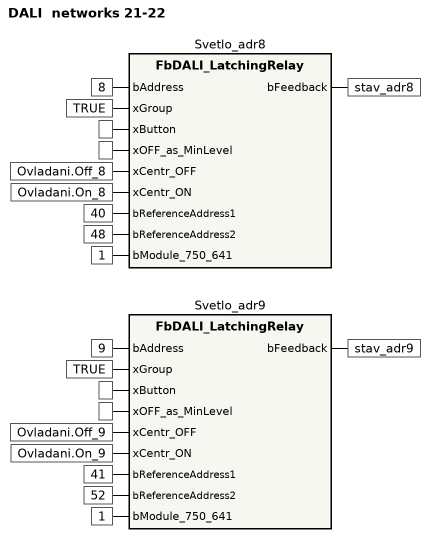
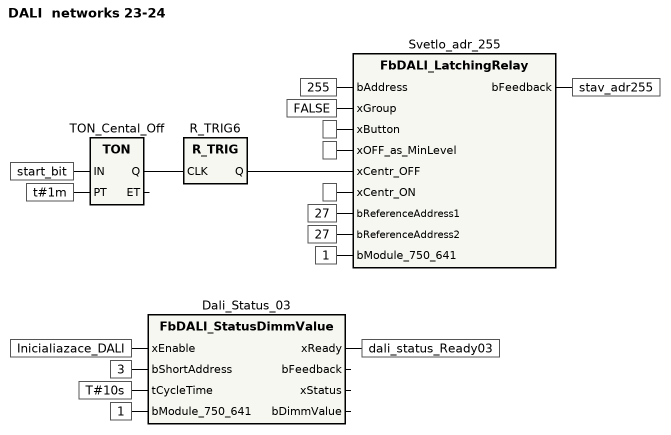
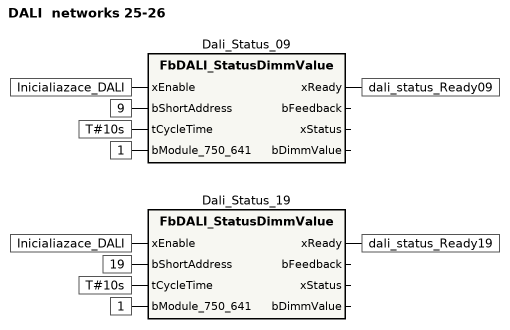
_FBD_ (* Function Block Diagram *)
NETWORK 1
	D_M:FbDALI_Joblist(bModule_750_641: 1)
NETWORK 2
	???:DALI_Config()
NETWORK 3
	Trojklik_Fagule_OUT13:Trojklik(TL1: , TL2: , TL3: , TL4: OR(TL10, TL10s, TL10p), TL5: , TL6: , RESET_Rezim_1klik: OR(OP_reset5, OP_reset1), RESET_Rezim_2klik: , RESET_Rezim_3klik: , RESET_Rezim_OUT15: , RESET_Rezim_OUT16: , Pocet_kliku_MAX: 1, AUT_vyp: FALSE, cas_vypnuti: t#30m, Rezim_1klik_OFF_ON => KA01, Rezim_OUT15_OFF_ON => KA13)
NETWORK 4
	ka13pink:TP(IN: ka13cas:TON(IN: KA13, PT: casvensvetel), PT: t#1s) => TL10p
NETWORK 5
	Fb_LatchingRelay1:Fb_LatchingRelay(Fb_ShortLong1:Fb_ShortLong(OR(TL06, TL06s, TL06p), 10, 1, 1, out 2 => KratkyKlikA), , , ) => KA15
NETWORK 6
	ka15pink:TP(IN: ka15cas:TON(IN: KA15, PT: casvensvetel), PT: t#1s) => TL06p
NETWORK 7
	Fb_LatchingRelay2:Fb_LatchingRelay(Fb_ShortLong2:Fb_ShortLong(OR(TL05, TL05s, TL04, TL05p), 10, 1, 1, out 2 => KratkyKlikB), , , ) => KA16
NETWORK 8
	ka16pink:TP(IN: ka16cas:TON(IN: KA16, PT: casvensvetel), PT: t#1s) => TL05p
NETWORK 9
	Fb_ShortLong3:Fb_ShortLong(OR(TL03, TL01, TL01s, TL02), 10, 1, 1, out 2 => KratkyKlikC)
NETWORK 10
	OR(KratkyKlikA, KratkyKlikB, KratkyKlikC) => KratkyKlik
NETWORK 11
	CTU1:CTU(CU: AND(TP1:TP(IN: KratkyKlik, PT: CasNaKlik), R_TRIG1:R_TRIG(CLK: KratkyKlik)), RESET: R_TRIG2:R_TRIG(CLK: Zhasni1.xPresunuto), PV: 3, CV => STAV)
NETWORK 12
	Zhasni1:Zhasni(wIn: STAV, xPresun: F_TRIG3:F_TRIG(CLK: TP1.Q))
NETWORK 13
	Svetlo_adr1:FbDALI_LatchingRelay(bAddress: 1, xGroup: TRUE, xButton: , xOFF_as_MinLevel: , xCentr_OFF: Zhasni1.xoffOUT1, xCentr_ON: Zhasni1.xonOUT1, bReferenceAddress1: 3, bReferenceAddress2: 9, bModule_750_641: 1) => stav_adr1
NETWORK 14
	Svetlo_adr2:FbDALI_LatchingRelay(bAddress: 2, xGroup: TRUE, xButton: , xOFF_as_MinLevel: , xCentr_OFF: Zhasni1.xoffOUT2, xCentr_ON: Zhasni1.xonOUT2, bReferenceAddress1: 17, bReferenceAddress2: 17, bModule_750_641: 1) => stav_adr2
NETWORK 15
	Svetlo_adr3:FbDALI_LatchingRelay(bAddress: 3, xGroup: TRUE, xButton: , xOFF_as_MinLevel: , xCentr_OFF: Zhasni1.xoffOUT3, xCentr_ON: Zhasni1.xonOUT3, bReferenceAddress1: 27, bReferenceAddress2: 27, bModule_750_641: 1) => stav_adr3
NETWORK 16
	Svetlo_adr4:FbDALI_DimmSingleButton(bAddress: 4, xGroup: TRUE, xButton: OR(TL09, TL09s), bSwitchOnLevel: hodnota_po_zapnuti_prodejna, xOFF_at_MinLevel: povolit_vypnuti_pri_minimum, xOFF_as_MinLevel: , bFadeRate: rychlost_zneny, tShortPushButton: co_je_kratky_a_dlouhy_stisk, bReferenceaddress1: 29, bReferenceaddress2: 30, bModule_750_641: 1) => stav_adr4
NETWORK 17
	Svetlo_adr5:FbDALI_LatchingRelay(bAddress: 5, xGroup: TRUE, xButton: OR(TL12, FALSE), xOFF_as_MinLevel: , xCentr_OFF: , xCentr_ON: , bReferenceAddress1: 37, bReferenceAddress2: 45, bModule_750_641: 1) => stav_adr5
NETWORK 18
	Svetlo_adr6:FbDALI_LatchingRelay(bAddress: 6, xGroup: TRUE, xButton: OR(TL13, FALSE), xOFF_as_MinLevel: , xCentr_OFF: , xCentr_ON: , bReferenceAddress1: 47, bReferenceAddress2: 49, bModule_750_641: 1) => stav_adr6
NETWORK 19
	Ovladani:Ovladani_7_8_9(xVstup: OR(TL11, FALSE), rCidlo: Cidlo, rUroven1: Uroven1, rUroven2: Uroven2, tZpozdeniCidla: DWORD_TO_TIME(MUL(ZpozdeniCidla, 60000)))
NETWORK 20
	Svetlo_adr7:FbDALI_LatchingRelay(bAddress: 7, xGroup: TRUE, xButton: , xOFF_as_MinLevel: , xCentr_OFF: Ovladani.Off_7, xCentr_ON: Ovladani.On_7, bReferenceAddress1: 36, bReferenceAddress2: 50, bModule_750_641: 1) => stav_adr7
NETWORK 21
	Svetlo_adr8:FbDALI_LatchingRelay(bAddress: 8, xGroup: TRUE, xButton: , xOFF_as_MinLevel: , xCentr_OFF: Ovladani.Off_8, xCentr_ON: Ovladani.On_8, bReferenceAddress1: 40, bReferenceAddress2: 48, bModule_750_641: 1) => stav_adr8
NETWORK 22
	Svetlo_adr9:FbDALI_LatchingRelay(bAddress: 9, xGroup: TRUE, xButton: , xOFF_as_MinLevel: , xCentr_OFF: Ovladani.Off_9, xCentr_ON: Ovladani.On_9, bReferenceAddress1: 41, bReferenceAddress2: 52, bModule_750_641: 1) => stav_adr9
NETWORK 23 (* Po 1min po restartu dojde k vypnuti vsech svitidel *)
	Svetlo_adr_255:FbDALI_LatchingRelay(bAddress: 255, xGroup: FALSE, xButton: , xOFF_as_MinLevel: , xCentr_OFF: R_TRIG6:R_TRIG(CLK: TON_Cental_Off:TON(IN: start_bit, PT: t#1m)), xCentr_ON: , bReferenceAddress1: 27, bReferenceAddress2: 27, bModule_750_641: 1) => stav_adr255
NETWORK 24
	Dali_Status_03:FbDALI_StatusDimmValue(xEnable: Inicialiazace_DALI, bShortAddress: 3, tCycleTime: T#10s, bModule_750_641: 1) => dali_status_Ready03
NETWORK 25
	Dali_Status_09:FbDALI_StatusDimmValue(xEnable: Inicialiazace_DALI, bShortAddress: 9, tCycleTime: T#10s, bModule_750_641: 1) => dali_status_Ready09
NETWORK 26
	Dali_Status_19:FbDALI_StatusDimmValue(xEnable: Inicialiazace_DALI, bShortAddress: 19, tCycleTime: T#10s, bModule_750_641: 1) => dali_status_Ready19
_END_FBD_
(* the same logic as Structured Text *)
(* Network 1 *)
D_M(bModule_750_641 := 1);
(* Network 2: see the listing above *)
(* Network 3: see the listing above *)
(* Network 4 *)
ka13cas(IN := KA13, PT := casvensvetel);
ka13pink(IN := ka13cas.Q, PT := t#1s);
TL10p := ka13pink.Q;
(* Network 5: see the listing above *)
(* Network 6 *)
ka15cas(IN := KA15, PT := casvensvetel);
ka15pink(IN := ka15cas.Q, PT := t#1s);
TL06p := ka15pink.Q;
(* Network 7: see the listing above *)
(* Network 8 *)
ka16cas(IN := KA16, PT := casvensvetel);
ka16pink(IN := ka16cas.Q, PT := t#1s);
TL05p := ka16pink.Q;
(* Network 9: see the listing above *)
(* Network 10 *)
KratkyKlik := KratkyKlikA OR KratkyKlikB OR KratkyKlikC;
(* Network 11 *)
TP1(IN := KratkyKlik, PT := CasNaKlik);
R_TRIG1(CLK := KratkyKlik);
R_TRIG2(CLK := Zhasni1.xPresunuto);
CTU1(CU := TP1.Q AND R_TRIG1.Q, RESET := R_TRIG2.Q, PV := 3);
STAV := CTU1.CV;
(* Network 12 *)
F_TRIG3(CLK := TP1.Q);
Zhasni1(wIn := STAV, xPresun := F_TRIG3.Q);
(* Network 13: see the listing above *)
(* Network 14: see the listing above *)
(* Network 15: see the listing above *)
(* Network 16: see the listing above *)
(* Network 17: see the listing above *)
(* Network 18: see the listing above *)
(* Network 19: see the listing above *)
(* Network 20: see the listing above *)
(* Network 21: see the listing above *)
(* Network 22: see the listing above *)
(* Network 23: see the listing above *)
(* Network 24 *)
Dali_Status_03(xEnable := Inicialiazace_DALI, bShortAddress := 3, tCycleTime := T#10s, bModule_750_641 := 1);
dali_status_Ready03 := Dali_Status_03.xReady;
(* Network 25 *)
Dali_Status_09(xEnable := Inicialiazace_DALI, bShortAddress := 9, tCycleTime := T#10s, bModule_750_641 := 1);
dali_status_Ready09 := Dali_Status_09.xReady;
(* Network 26 *)
Dali_Status_19(xEnable := Inicialiazace_DALI, bShortAddress := 19, tCycleTime := T#10s, bModule_750_641 := 1);
dali_status_Ready19 := Dali_Status_19.xReady;
END_PROGRAM

(* POU dali/Trojklik, FBD *)
FUNCTION_BLOCK Trojklik
VAR
	TLx_sklad: BOOL;
	Data_platna: BOOL;
	Data_platna_reset: BOOL;
	T_Data_platna: TON;
	T_Data_platna_reset: TON;
	Stisk_kratky: BOOL := FALSE;
	Stisk_dlouhy: BOOL := FALSE;
	Q_stisk_TLx: BOOL;
	T_stisk_TLx: TON;
	F_trig_hr1: F_TRIG;
	R_trig_hr2: R_TRIG;
	TLx_sklad_hr1: BOOL;
	TLx_INT: INT;
	TLx_Citac: CTU;
	SET_stisk_TLx: BOOL;
	SR_stisk_TLx: SR;

	ZAP_VYP_sklad: BOOL;
	mod_1klik: BOOL;
	mod_2klik: BOOL;
	blok: BOOL;
	blok_ZAP_VYP: BOOL;
	T_blok: TON;
	T_blok_ZAP_VYP: TON;
	TP_mode_1klik: TP;

	TP_mode_2klik: TP;

	TP_byl_kratky: TP;
	Q_byl_kratky: BOOL;
	blok_kratky: BOOL;
	mod_3klik: BOOL;
	TP_mode_3klik: TP;

	TP_reset1: TP;
	TP_reset2: TP;
	TP_reset3: TP;
	TLx_zvenku: BOOL;
	T_stisk_TLx_zvenku: TON;
	TLx_sklad_hr1_zvenku: BOOL;
	F_trig_hr1_zvenku: F_TRIG;
	Stisk_kratky_zvenku: BOOL;
	SET_stisk_TLx_zvenku: BOOL;
	Q_byl_kratky_zvenku: BOOL;
	TP_byl_kratky_zvenku: TP;
	Stisk_dlouhy_zvenku: BOOL;
	blok_kratky_zvenku: BOOL;
	TLx_INT_zvenku: INT;
	TLx_Citac_zvenku: CTU;
	Q_stisk_TLx_zvenku: BOOL;
	R_trig_hr2_zvenku: R_TRIG;
	SR_stisk_TLx_zvenku: SR;
	blok_OUT15: BOOL;
	TOF_OUT15_zp: TOF;
	R_trig_OUT15: R_TRIG;
	R_trig_OUT15b: R_TRIG;
	TON_blok_OUT15: TON;
	TON_AUT_stop_OUT15: TON;
	R_trig_OUT16: R_TRIG;
	TOF_OUT16_zp: TOF;
	blok_OUT16: BOOL;
	R_trig_OUT16b: R_TRIG;
	TON_AUT_stop_OUT16: TON;
	TON_blok_OUT16: TON;
	T_max: TON;
	Q_T_MAX: BOOL;
	TP_T_max: TP;
	Aktivni_TL1: BOOL;
	Aktivni_TL2: BOOL;
	Aktivni_TL3: BOOL;
	Aktivni_TL4: BOOL;
	Aktivni_TL5: BOOL;
	Aktivni_TL6: BOOL;
	T_vypnuti_ukonceno: TP;
	Q_vypnuti_ukonceno: BOOL;
	F_trig_1klik: F_TRIG;
	F_trig_2klik: F_TRIG;
	F_trig_3klik: F_TRIG;
	tp_1klik_vyp: TP;
	f_trig_1klik_vyp: F_TRIG;
	tp_2klik_vyp: TP;
	f_trig_2klik_vyp: F_TRIG;
	f_trig_3klik_vyp: F_TRIG;
	tp_3klik_vyp: TP;
END_VAR

VAR_OUTPUT
	Rezim_1klik_PULS: BOOL;
	Rezim_1klik_OFF_ON: BOOL;
	Rezim_2klik_PULS: BOOL;
	Rezim_2klik_OFF_ON: BOOL;
	Rezim_3klik_PULS: BOOL;
	Rezim_3klik_OFF_ON: BOOL;
	Rezim_OUT15_OFF_ON: BOOL;
	Rezim_OUT16_OFF_ON: BOOL;
END_VAR
VAR_INPUT
	TL1: BOOL;
	TL2: BOOL;
	TL3: BOOL;
	TL4: BOOL;
	TL5: BOOL;
	TL6: BOOL;
	RESET_Rezim_1klik: BOOL;
	RESET_Rezim_2klik: BOOL;
	RESET_Rezim_3klik: BOOL;
	RESET_Rezim_OUT15: BOOL;
	RESET_Rezim_OUT16: BOOL;
	Pocet_kliku_MAX: INT;
	AUT_vyp: BOOL;
	cas_vypnuti: TIME;
END_VAR
VAR (* helpers for the ST form of the networks *)
	_p1 : BOOL;
	_p2 : BOOL;
	_p3 : BOOL;
	_p4 : BOOL;
	_p5 : BOOL;
	_p6 : BOOL;
	_p7 : BOOL;
END_VAR
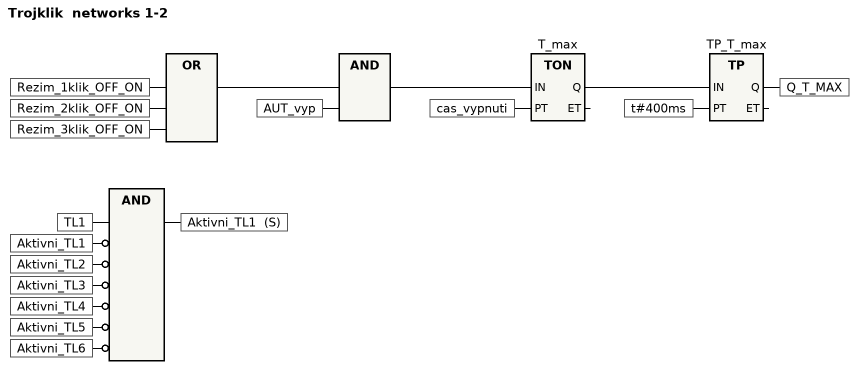
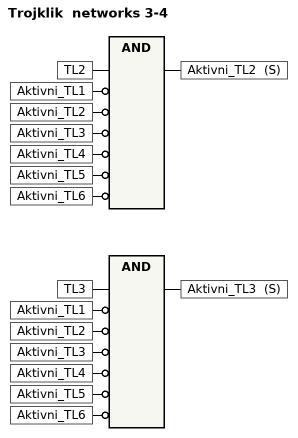
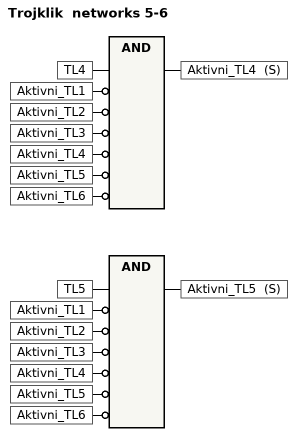
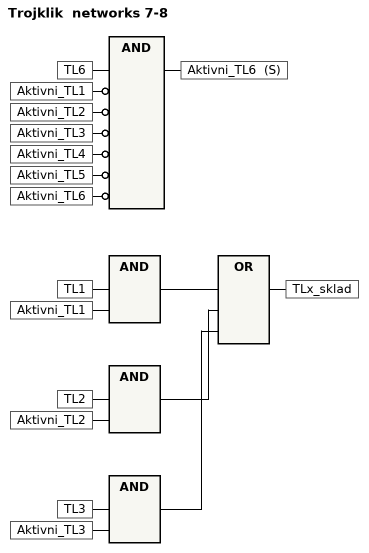
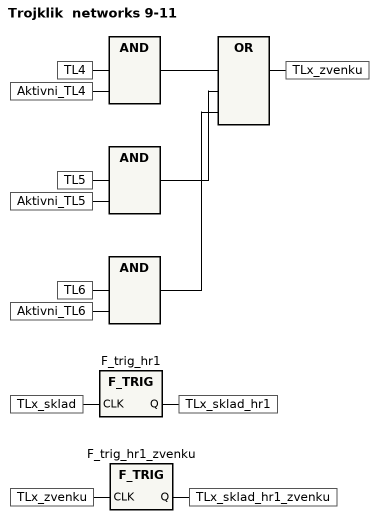
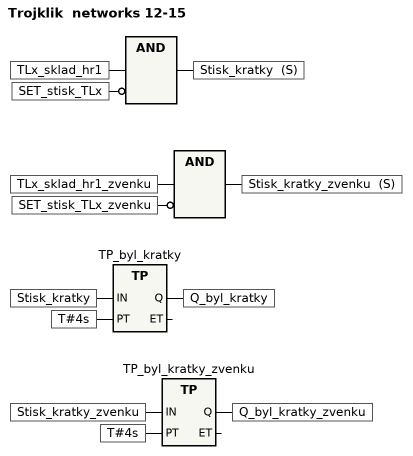
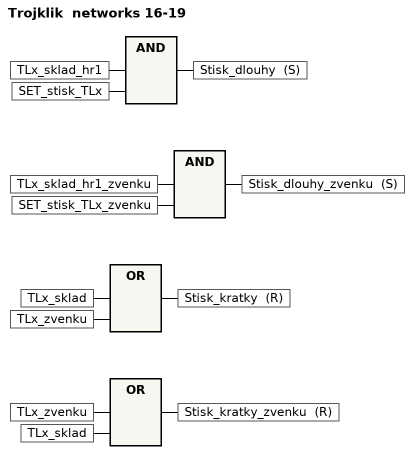
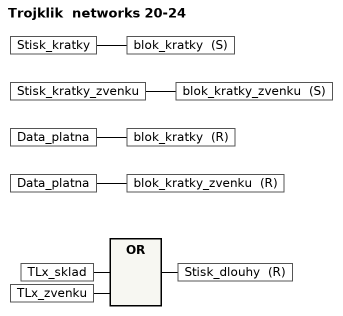
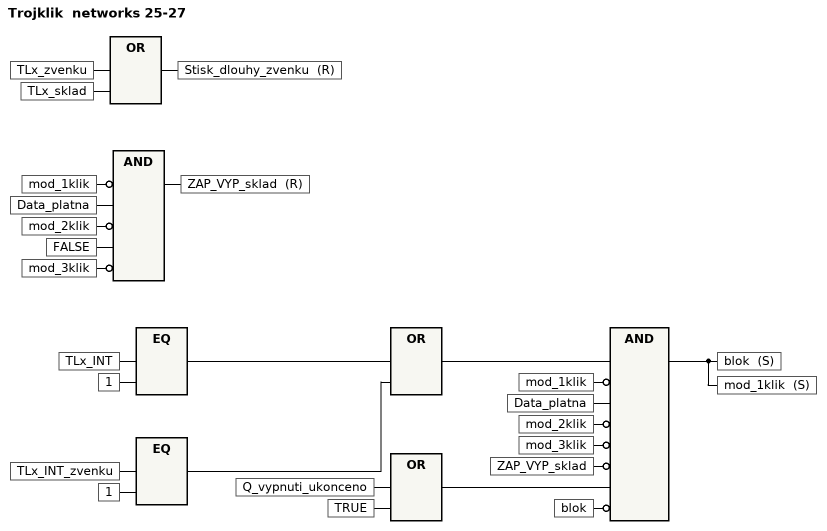
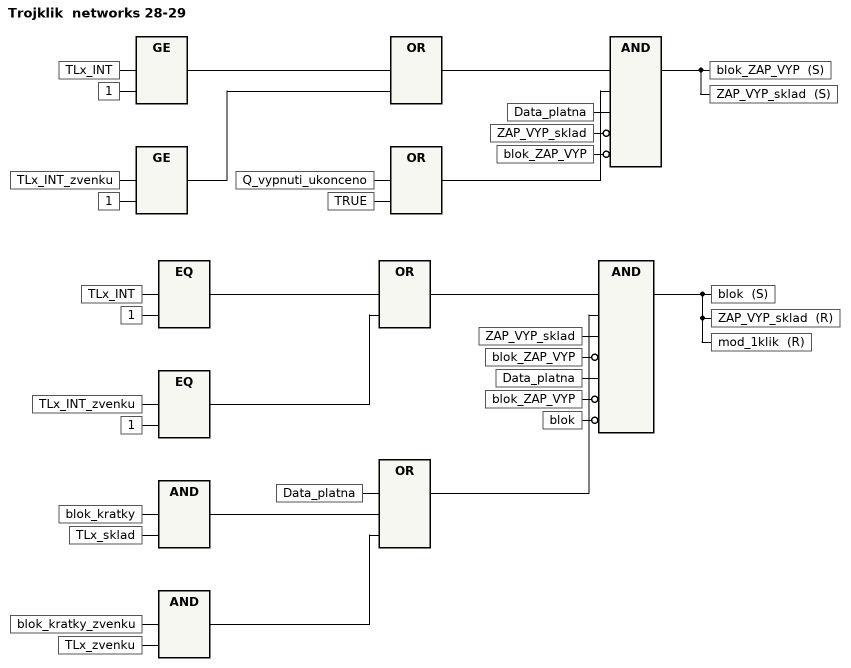
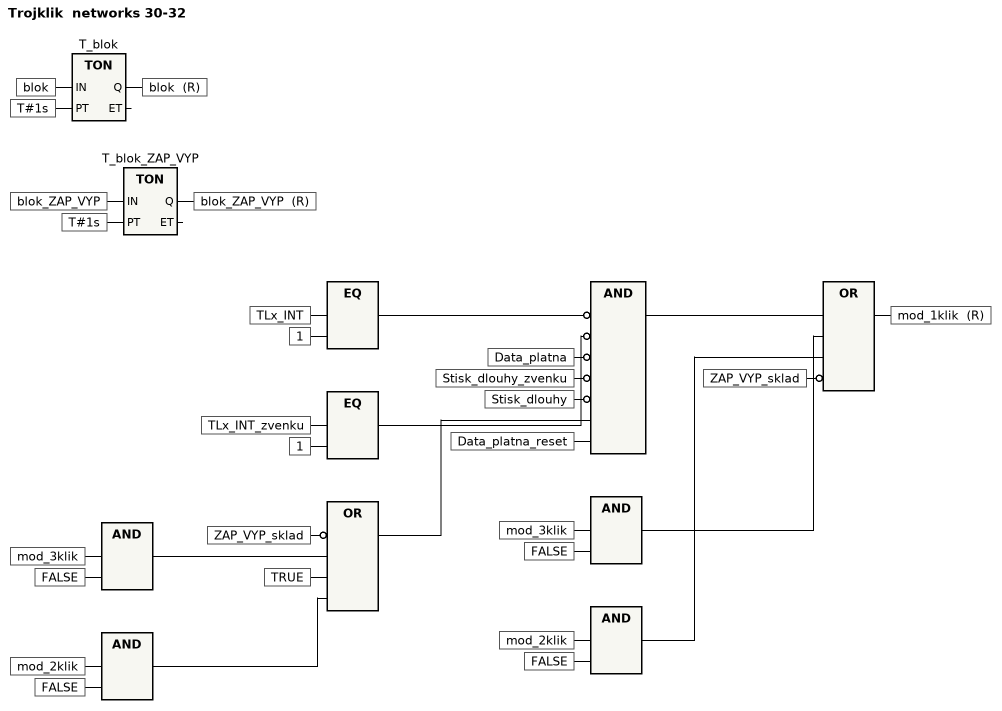
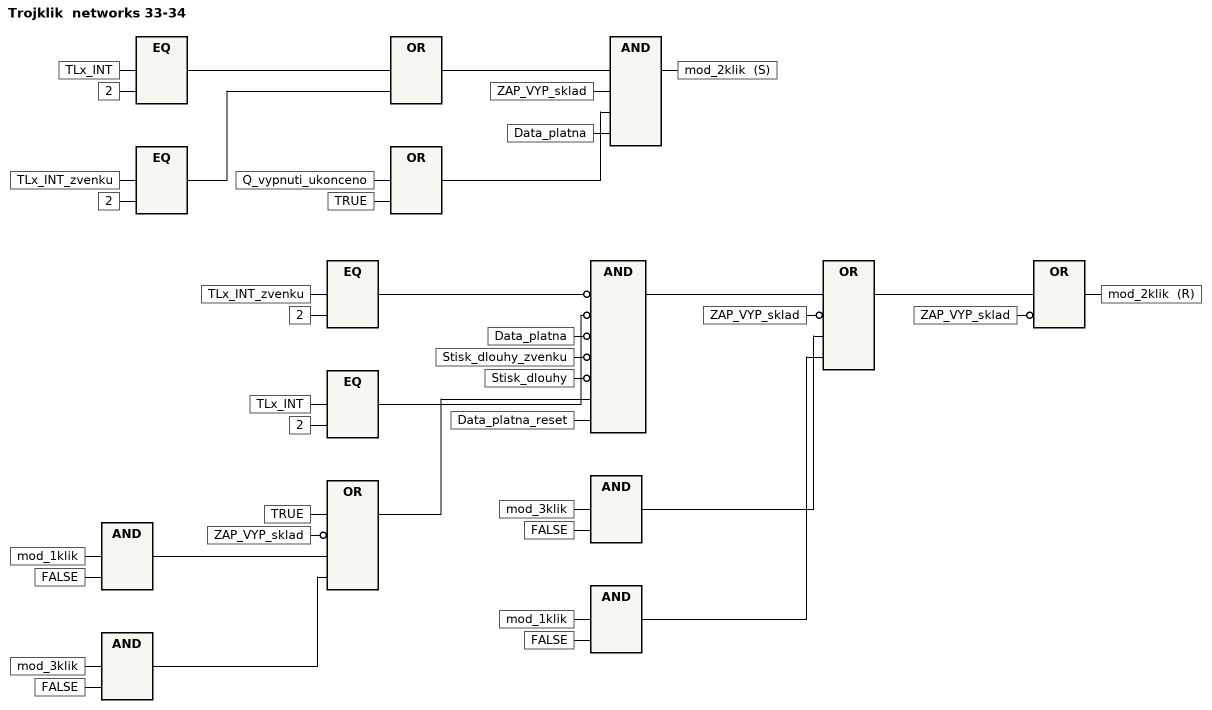
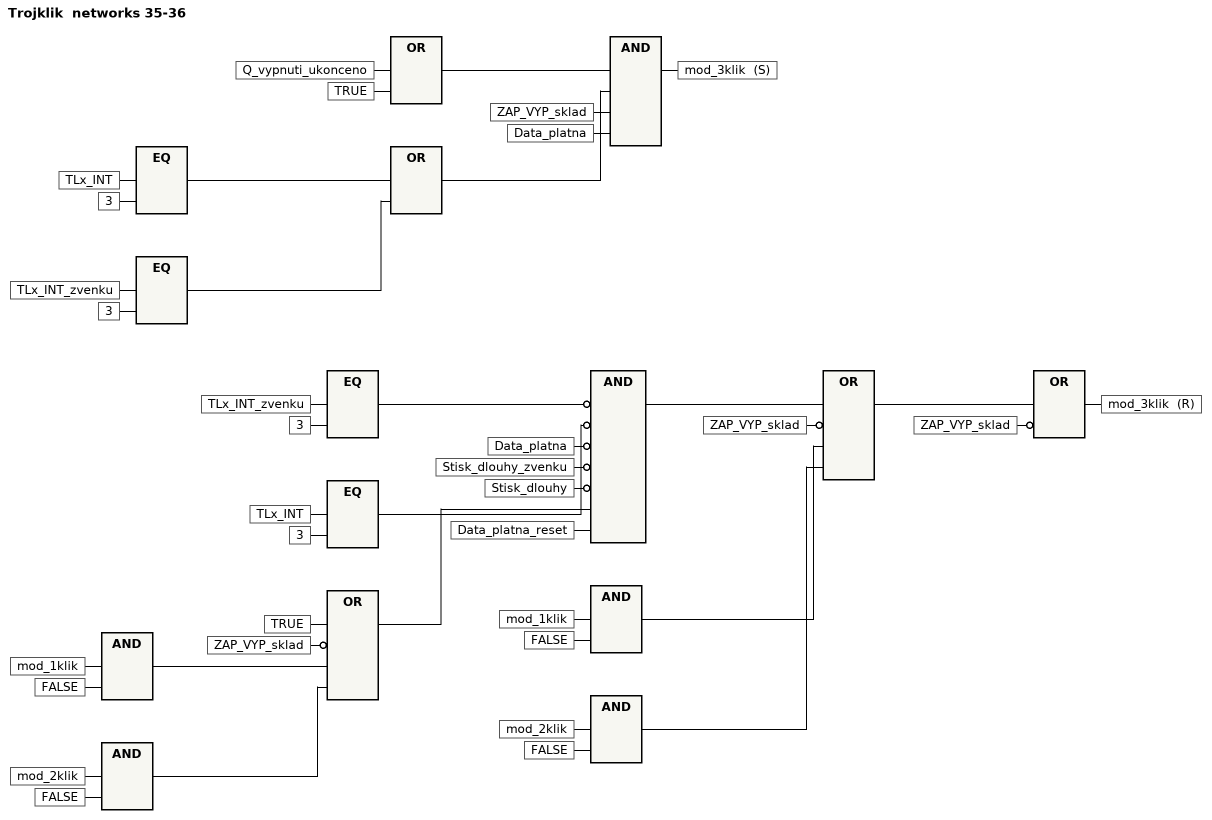
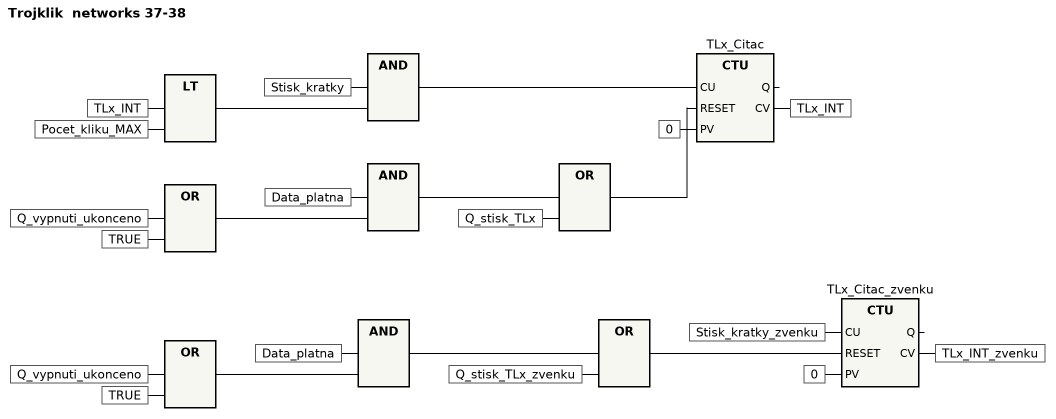
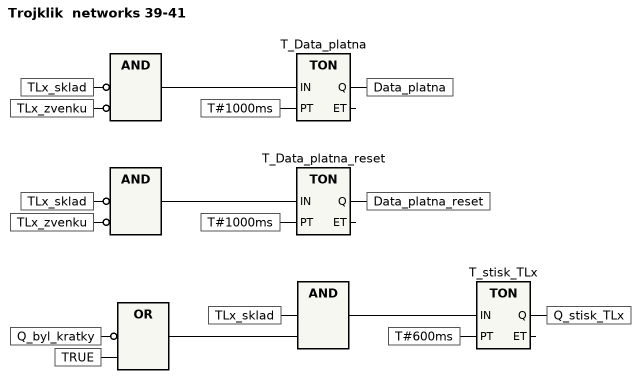
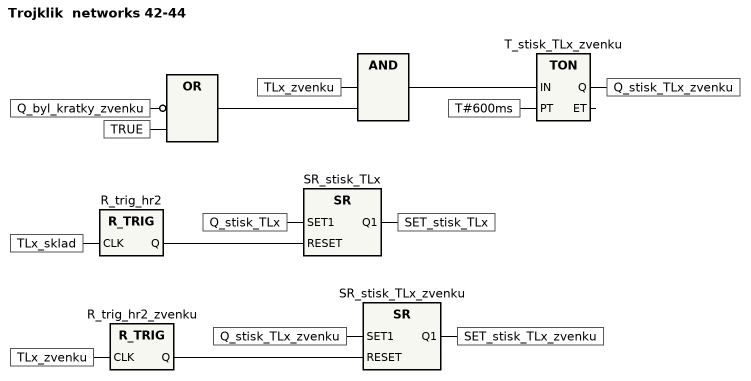
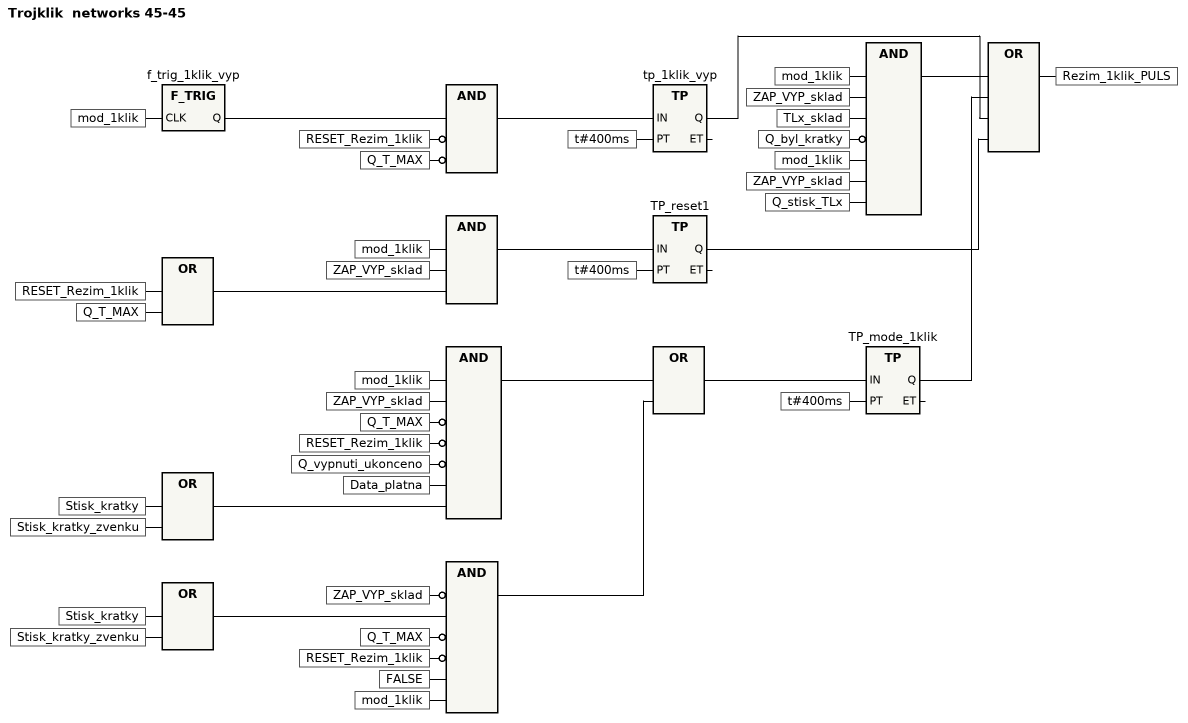
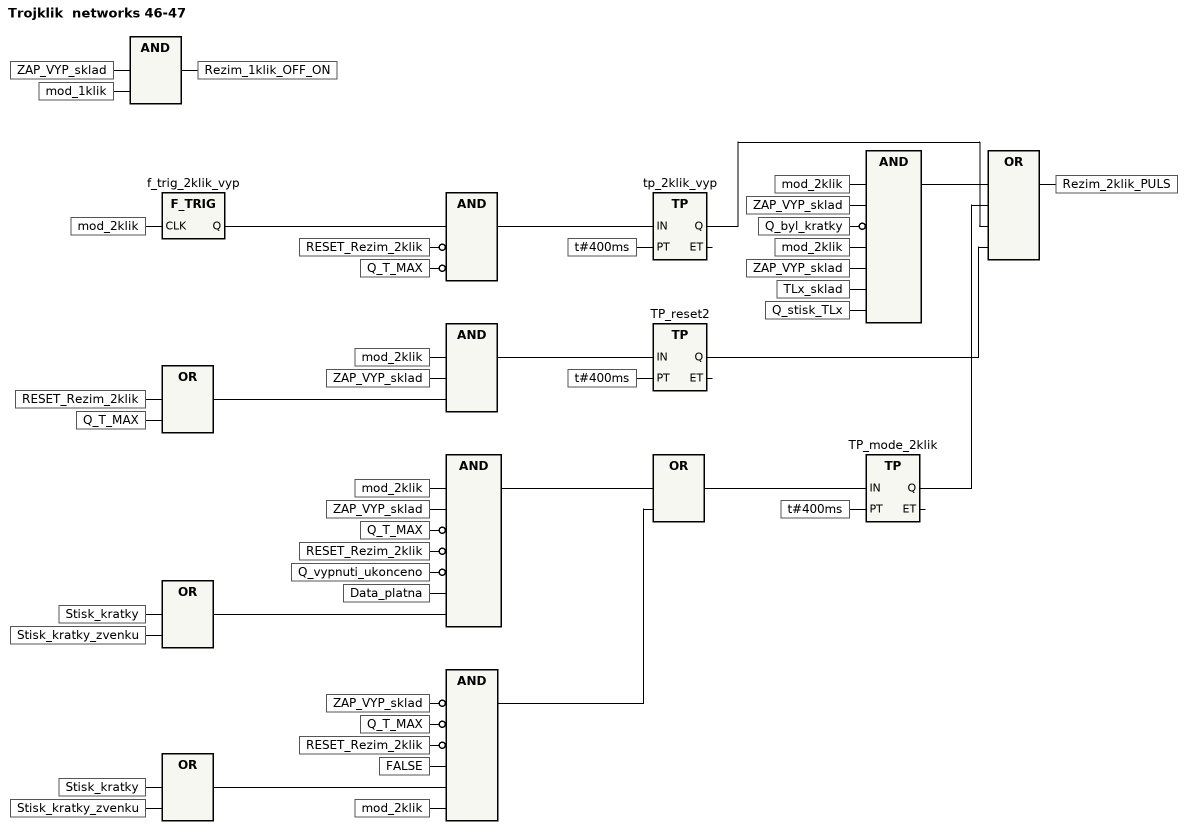
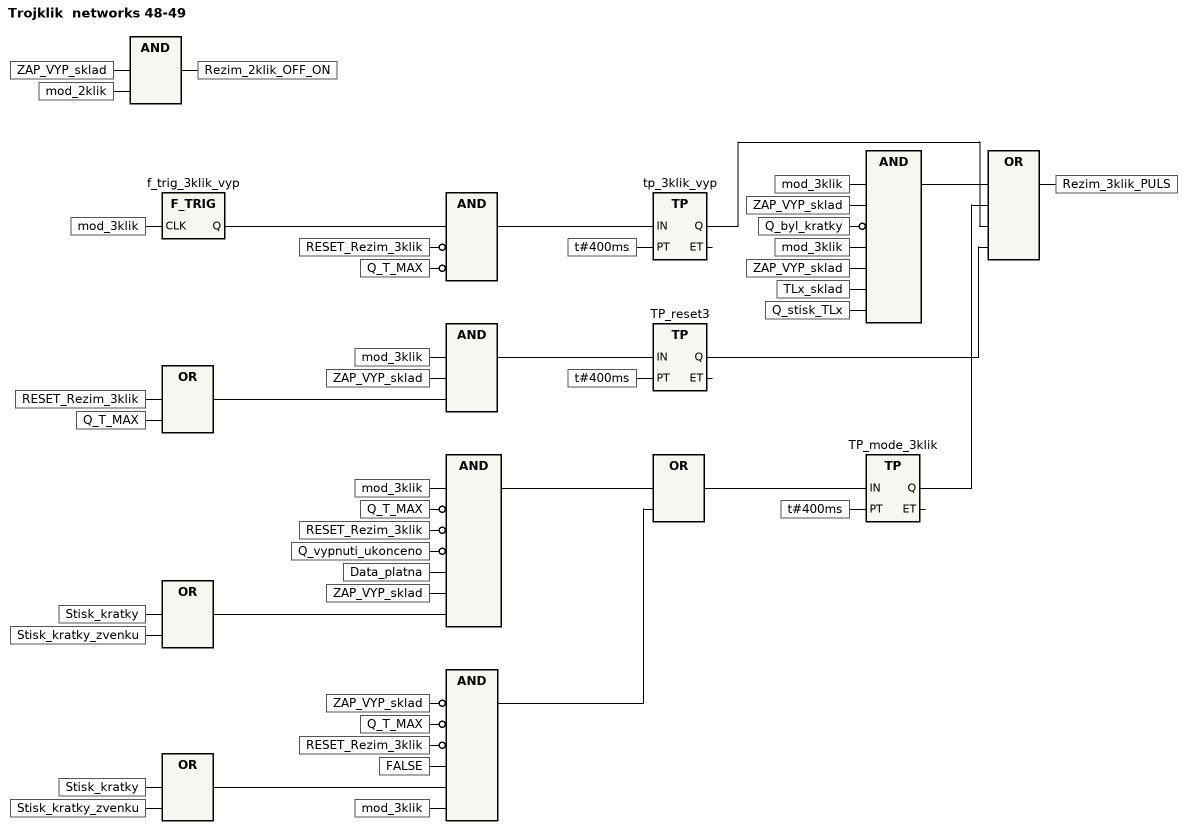
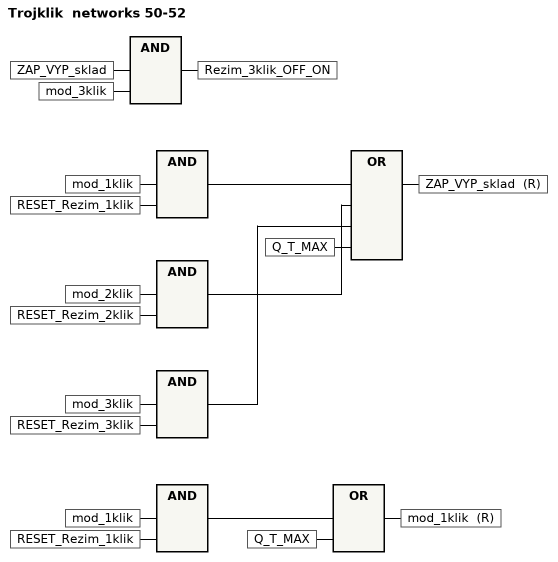
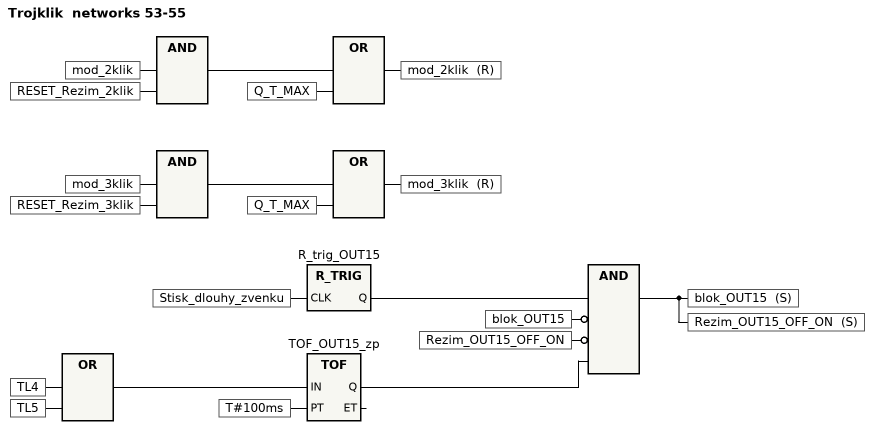
